PROGRAM MAIN
VAR
END_VAR

Motor_Control();

END_PROGRAM

(* stored: Version 1.1.0.1, ProductVersion 3.1.4024.12
   POU MAIN: Id {735f8b3b-db36-4fe1-a63b-8fcf7a0ed59f}, SpecialFunc None *)
